FUNCTION_BLOCK CylinderTestContext EXTENDS TcoCore._internals_TcoContext
VAR
	{attribute addProperty _moveHomeDefaultName "<#MOVE HOME SWEET HOME#>"}
	{attribute addProperty _moveWorkDefaultName "<#MOVE TO WORK HARD WORK#>"}
	{attribute addProperty _stopDefaultName "<#STOP AND THINK#>"}
	_sut			: TcoPneumatics.TcoCylinder(THIS^);
	_sutInvalid 	: TcoPneumatics.TcoCylinder(THIS^);
	_atHomeSignal	: BOOL;
	_moveHomeSignal : BOOL;
	_atWorkSignal	: BOOL;
	_moveWorkSignal : BOOL;
END_VAR
VAR
	_moveHomeDone	: BOOL;
	_moveWorkDone : BOOL;	
	_disableSignal : BOOL;
END_VAR

METHOD PROTECTED Main

_sut(inoAtHomePos := _atHomeSignal,
    inoAtWorkPos := _atWorkSignal,
    inoToHomePos := _moveHomeSignal,
    inoToWorkPos := _moveWorkSignal);

CASE _testId OF
	eCyclinderTests.Invalid:
	_sutInvalid.Stop();
	_sutInvalid.MoveToHome();
	_sutInvalid.MoveToWork();
	_sutInvalid.Service();
	_sutInvalid.AtHome;
	_sutInvalid.AtWork;
	_sutInvalid.AbortMoveHome(_disableSignal);
	_sutInvalid.AbortMoveHome(_disableSignal);
    eCyclinderTests.StopMovement:
        _sut.Stop();
    eCyclinderTests.MoveHomeMoving:
        _moveHomeDone := _sut.MoveToHome().Done;
    eCyclinderTests.MoveHomeMovingReached:
        _moveHomeDone := _sut.MoveToHome().Done;
    eCyclinderTests.MoveWorkMoving:
        _moveWorkDone := _sut.MoveToWork().Done;
    eCyclinderTests.MoveWorkMovingReached:
        _moveWorkDone := _sut.MoveToWork().Done;
    eCyclinderTests.AbortMoveTask:
        _sut.MoveHomeTask.Abort();	
	eCyclinderTests.DisableHome:
        _sut.AbortMoveHome(_disableSignal);
	eCyclinderTests.DisableWork:
        _sut.AbortMoveWork(_disableSignal);		
END_CASE
END_METHOD

END_FUNCTION_BLOCK

(* stored: Version 1.1.0.1, ProductVersion 3.1.4024.9
   POU CylinderTestContext: Id {4f0e4024-4378-058d-21b2-dd1a5c077cb8}, SpecialFunc None
   Method Main: Id {d7464bf3-4a73-0bd9-1c20-65d4ea0101c4} *)
